Fanuc KAREL source: kt00378.KL

-- PROVISIONAL review KL for V770-1; original PC SHA256 f3eab960e4b675ecac55d81c6f937451d93651563dbb46205e2b9b2467520933
-- Incomplete behavior may be omitted. Consult companion uncertainty JSON. Do not deploy.
PROGRAM KT00378
%NOLOCKGROUP
VAR
  OUT : BOOLEAN
-- UNRESOLVED_DECL Y1 type=002018
-- UNRESOLVED_DECL H2 type=002017
BEGIN
  -- UNRESOLVED_PC offsets 5-19; opcodes 2E,22,9D,33,B2
  -- UNRESOLVED_PC offsets 24-38; opcodes 2E,22,9D,33,B4
  -- UNRESOLVED_PC offsets 43-68; opcodes 22,9D,33,B1,22,9D,33,B3,5A,23
  -- UNRESOLVED_PC offsets 73-77; opcodes 7F
END KT00378
